// TIA Portal project "项目3" (V15)

(* hardware
DEVICE "S7-1200 station_1"  S7-1200 Station
   slot 0: "Rack_0"  S7-1200 Rack  Rack  V1.0
   slot 1: "PLC_1"  CPU 1214C DC/DC/Rly  6ES7 214-1HG40-0XB0  V4.2
DEVICE "HMI_1"  TP1500 Comfort Outdoor
   slot 0: "HMI_1"  TP1500 Comfort Outdoor  6AV2 124-0QC13-0AX0  15.0.0.0
   slot 1: "HMI_RT_1"  TP1500 Comfort Outdoor  6AV2 124-0QC13-0AX0  15.0.0.0
   slot 5: "HMI_1.IE_CP_1"  PROFINET Interface  15.0.0.0
      slot 1: "PROFINET Interface_1"  PROFINET Interface
         slot 1: "Port_1"  Port
         slot 2: "Port_2"  Port
   slot 7: "HMI_1.MPI/DP_CP_1"  MPI/DP Interface  15.0.0.0
*)

// ===== PLC "PLC_1"  CPU 1214C DC/DC/Rly =====

VAR_GLOBAL   // PLC tag table "默认变量表"
   "东西绿" AT %Q12.0 : Bool;
   "东西黄" AT %Q12.1 : Bool;
   "东西红" AT %Q12.2 : Bool;
   "东西转向" AT %Q12.3 : Bool;
   "南北绿" AT %Q12.4 : Bool;
   "南北黄" AT %Q12.5 : Bool;
   "南北红" AT %Q12.6 : Bool;
   "南北转向" AT %Q12.7 : Bool;
   "启动" AT %I4.0 : Bool;
   "System_Byte" AT %MB1 : Byte;
   "FirstScan" AT %M1.0 : Bool;
   "DiagStatusUpdate" AT %M1.1 : Bool;
   "AlwaysTRUE" AT %M1.2 : Bool;
   "AlwaysFALSE" AT %M1.3 : Bool;
   "Clock_Byte" AT %MB0 : Byte;
   "Clock_10Hz" AT %M0.0 : Bool;
   "Clock_5Hz" AT %M0.1 : Bool;
   "Clock_2.5Hz" AT %M0.2 : Bool;
   "Clock_2Hz" AT %M0.3 : Bool;
   "Clock_1.25Hz" AT %M0.4 : Bool;
   "Clock_1Hz" AT %M0.5 : Bool;
   "Clock_0.625Hz" AT %M0.6 : Bool;
   "Clock_0.5Hz" AT %M0.7 : Bool;
   "Tag_1" AT %MD100 : Time;
   "data" AT %MD50 : DInt;
   "计数器输出" AT %MD54 : DInt;
   "计数器复位" AT %MD58 : DInt;
   "Tag_2" AT %Q10.0 : Bool;
   "东西红启动" AT %M3.0 : Bool;
   "南北转向启动" AT %M3.1 : Bool;
   "南北转向闪烁启动" AT %M3.2 : Bool;
   "南北绿启动" AT %M3.3 : Bool;
   "南北闪烁启动" AT %M3.4 : Bool;
   "南北黄启动" AT %M3.5 : Bool;
   "南北红启动" AT %M3.6 : Bool;
   "东西转向启动" AT %M3.7 : Bool;
   "东西转向闪烁启动" AT %M4.0 : Bool;
   "东西绿启动" AT %M4.1 : Bool;
   "东西闪烁启动" AT %M4.2 : Bool;
   "东西黄启动" AT %M4.3 : Bool;
   "停止" AT %I4.1 : Bool;
   "启动信号1" AT %Q5.7 : Bool;
   "定时器1当前值" AT %MD4 : DInt;
   "定时器2当前值" AT %MD5 : DInt;
   "定时器1输出" AT %Q5.0 : Bool;
   "定时器2输出" AT %Q5.1 : Bool;
   "正常信号" AT %Q5.2 : Bool;
   "高峰信号" AT %Q5.3 : Bool;
   "夜间信号" AT %Q5.4 : Bool;
   "启动信号2" AT %Q5.5 : Bool;
   "启动信号3" AT %Q5.6 : Bool;
   "时间" AT %MD20 : Time_Of_Day;
   "报警信号" AT %Q13.0 : Bool;
   "夜间手动" AT %I4.4 : Bool;
   "正常手动" AT %I4.5 : Bool;
   "高峰手动" AT %I4.6 : Bool;
   "手动信号" AT %M6.0 : Bool;
   "切换手动" AT %I4.2 : Bool;
   "切换自动" AT %I4.3 : Bool;
   "报警" AT %Q1.7 : Bool;
   "1" AT %Q2.0 : Bool;
   "2" AT %Q2.1 : Bool;
   "3" AT %Q2.2 : Bool;
END_VAR

DATA_BLOCK "系统时间"   // DB1
{ S7_Optimized_Access := 'TRUE' }
VERSION : 0.1
   VAR
      当前时间 : DTL;
      ret : Int;
      设定时间 : DTL;
      ret1 : Int;
      设定时间按钮 : Bool;
   END_VAR
BEGIN
END_DATA_BLOCK

DATA_BLOCK "夜间_DB"   // DB3
{ S7_Optimized_Access := 'TRUE' }
VERSION : 0.1
// stored: InstanceOfName 夜间
"夜间"
BEGIN
END_DATA_BLOCK

DATA_BLOCK "夜间_DB_1"   // DB4
{ S7_Optimized_Access := 'TRUE' }
VERSION : 0.1
// stored: InstanceOfName 夜间
"夜间"
BEGIN
END_DATA_BLOCK

DATA_BLOCK "高峰_DB_1"   // DB6
{ S7_Optimized_Access := 'TRUE' }
VERSION : 0.1
// stored: InstanceOfName 高峰
"高峰"
BEGIN
END_DATA_BLOCK

DATA_BLOCK "正常_DB_2"   // DB8
{ S7_Optimized_Access := 'TRUE' }
VERSION : 0.1
// stored: InstanceOfName 正常
"正常"
BEGIN
END_DATA_BLOCK

// folder: System blocks/Program resources

DATA_BLOCK "计数器"   // DB2
{ S7_Optimized_Access := 'TRUE' }
AUTHOR : Simatic
FAMILY : IEC
NAME : CNTR
VERSION : 1.0
// stored: InstanceOfName IEC_COUNTER
"IEC_COUNTER"
BEGIN
END_DATA_BLOCK

DATA_BLOCK "IEC_Timer_0_DB_2"   // DB10
{ S7_Optimized_Access := 'TRUE' }
AUTHOR : Simatic
FAMILY : IEC
NAME : IEC_TMR
VERSION : 1.0
// stored: InstanceOfName IEC_TIMER
"IEC_TIMER"
BEGIN
END_DATA_BLOCK

DATA_BLOCK "IEC_Timer_0_DB_3"   // DB11
{ S7_Optimized_Access := 'TRUE' }
AUTHOR : Simatic
FAMILY : IEC
NAME : IEC_TMR
VERSION : 1.0
// stored: InstanceOfName IEC_TIMER
"IEC_TIMER"
BEGIN
END_DATA_BLOCK

// folder: (top level)

FUNCTION_BLOCK "正常"   // FB1, LAD
{ S7_Optimized_Access := 'TRUE' }
VERSION : 0.1
   VAR_INPUT
      启动 : Bool;
   END_VAR
   VAR_OUTPUT
      东西红 : Bool;
      南北转向 : Bool;
      南北绿 : Bool;
      南北黄 : Bool;
      南北红 : Bool;
      东西转向 : Bool;
      东西绿 : Bool;
      东西黄 : Bool;
   END_VAR
BEGIN

REGION Network 1: 计数
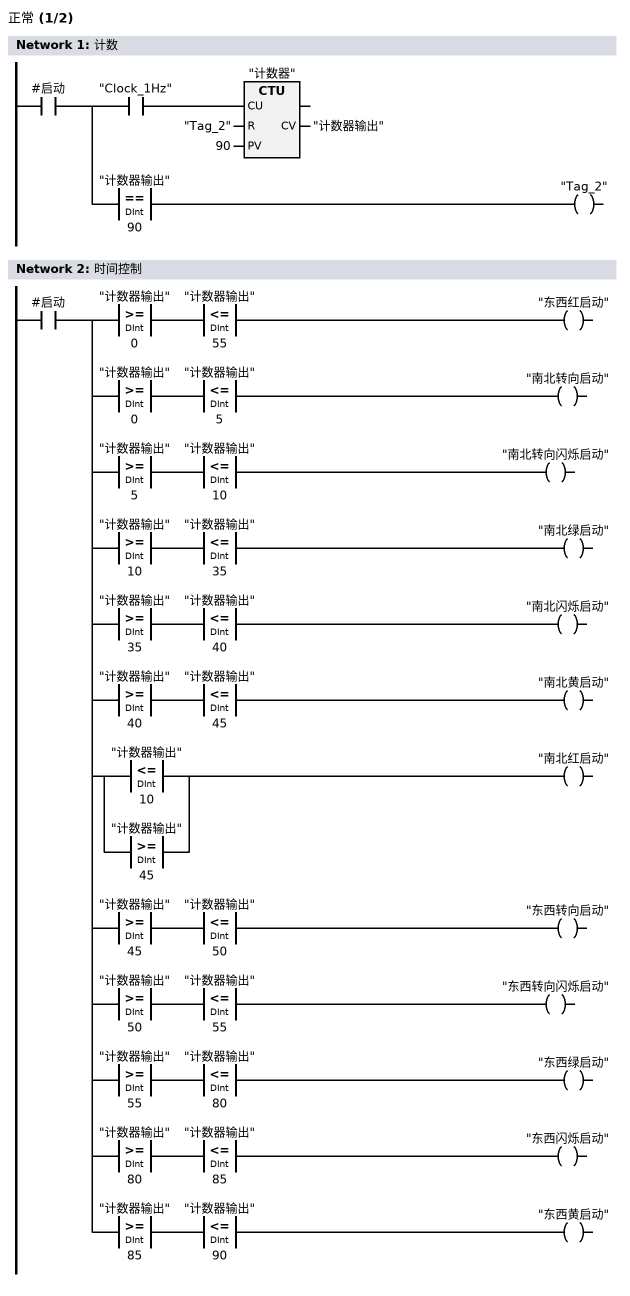
   "计数器".CTU(CU := #启动 AND "Clock_1Hz", R := "Tag_2", PV := 90, CV => "计数器输出");
   "Tag_2" := #启动 AND ("计数器输出" = 90);
END_REGION

REGION Network 2: 时间控制
   RUNG wire#powerrail
      Contact( #启动 )
      wire#w1
      { S7_Templates := "SrcType := DInt" } GE_Contact(in1 := "计数器输出", in2 := 0)
      { S7_Templates := "SrcType := DInt" } LE_Contact(in1 := "计数器输出", in2 := 55)
      Coil( "东西红启动" )
   END_RUNG
   RUNG wire#w1
      { S7_Templates := "SrcType := DInt" } GE_Contact(in1 := "计数器输出", in2 := 0)
      { S7_Templates := "SrcType := DInt" } LE_Contact(in1 := "计数器输出", in2 := 5)
      Coil( "南北转向启动" )
   END_RUNG
   RUNG wire#w1
      { S7_Templates := "SrcType := DInt" } GE_Contact(in1 := "计数器输出", in2 := 5)
      { S7_Templates := "SrcType := DInt" } LE_Contact(in1 := "计数器输出", in2 := 10)
      Coil( "南北转向闪烁启动" )
   END_RUNG
   RUNG wire#w1
      { S7_Templates := "SrcType := DInt" } GE_Contact(in1 := "计数器输出", in2 := 10)
      { S7_Templates := "SrcType := DInt" } LE_Contact(in1 := "计数器输出", in2 := 35)
      Coil( "南北绿启动" )
   END_RUNG
   RUNG wire#w1
      { S7_Templates := "SrcType := DInt" } GE_Contact(in1 := "计数器输出", in2 := 35)
      { S7_Templates := "SrcType := DInt" } LE_Contact(in1 := "计数器输出", in2 := 40)
      Coil( "南北闪烁启动" )
   END_RUNG
   RUNG wire#w1
      { S7_Templates := "SrcType := DInt" } GE_Contact(in1 := "计数器输出", in2 := 40)
      { S7_Templates := "SrcType := DInt" } LE_Contact(in1 := "计数器输出", in2 := 45)
      Coil( "南北黄启动" )
   END_RUNG
   RUNG wire#w1
      { S7_Templates := "SrcType := DInt" } LE_Contact(in1 := "计数器输出", in2 := 10)
      wire#w2
      Coil( "南北红启动" )
   END_RUNG
   RUNG wire#w1
      { S7_Templates := "SrcType := DInt" } GE_Contact(in1 := "计数器输出", in2 := 45)
   END_RUNG wire#w2
   RUNG wire#w1
      { S7_Templates := "SrcType := DInt" } GE_Contact(in1 := "计数器输出", in2 := 45)
      { S7_Templates := "SrcType := DInt" } LE_Contact(in1 := "计数器输出", in2 := 50)
      Coil( "东西转向启动" )
   END_RUNG
   RUNG wire#w1
      { S7_Templates := "SrcType := DInt" } GE_Contact(in1 := "计数器输出", in2 := 50)
      { S7_Templates := "SrcType := DInt" } LE_Contact(in1 := "计数器输出", in2 := 55)
      Coil( "东西转向闪烁启动" )
   END_RUNG
   RUNG wire#w1
      { S7_Templates := "SrcType := DInt" } GE_Contact(in1 := "计数器输出", in2 := 55)
      { S7_Templates := "SrcType := DInt" } LE_Contact(in1 := "计数器输出", in2 := 80)
      Coil( "东西绿启动" )
   END_RUNG
   RUNG wire#w1
      { S7_Templates := "SrcType := DInt" } GE_Contact(in1 := "计数器输出", in2 := 80)
      { S7_Templates := "SrcType := DInt" } LE_Contact(in1 := "计数器输出", in2 := 85)
      Coil( "东西闪烁启动" )
   END_RUNG
   RUNG wire#w1
      { S7_Templates := "SrcType := DInt" } GE_Contact(in1 := "计数器输出", in2 := 85)
      { S7_Templates := "SrcType := DInt" } LE_Contact(in1 := "计数器输出", in2 := 90)
      Coil( "东西黄启动" )
   END_RUNG
   // the same network as SCL:
   "东西红启动" := #启动 AND ("计数器输出" >= 0) AND ("计数器输出" <= 55);
   "南北转向启动" := #启动 AND ("计数器输出" >= 0) AND ("计数器输出" <= 5);
   "南北转向闪烁启动" := #启动 AND ("计数器输出" >= 5) AND ("计数器输出" <= 10);
   "南北绿启动" := #启动 AND ("计数器输出" >= 10) AND ("计数器输出" <= 35);
   "南北闪烁启动" := #启动 AND ("计数器输出" >= 35) AND ("计数器输出" <= 40);
   "南北黄启动" := #启动 AND ("计数器输出" >= 40) AND ("计数器输出" <= 45);
   "南北红启动" := #启动 AND (("计数器输出" <= 10) OR ("计数器输出" >= 45));
   "东西转向启动" := #启动 AND ("计数器输出" >= 45) AND ("计数器输出" <= 50);
   "东西转向闪烁启动" := #启动 AND ("计数器输出" >= 50) AND ("计数器输出" <= 55);
   "东西绿启动" := #启动 AND ("计数器输出" >= 55) AND ("计数器输出" <= 80);
   "东西闪烁启动" := #启动 AND ("计数器输出" >= 80) AND ("计数器输出" <= 85);
   "东西黄启动" := #启动 AND ("计数器输出" >= 85) AND ("计数器输出" <= 90);
END_REGION

REGION Network 3: 信号灯控制
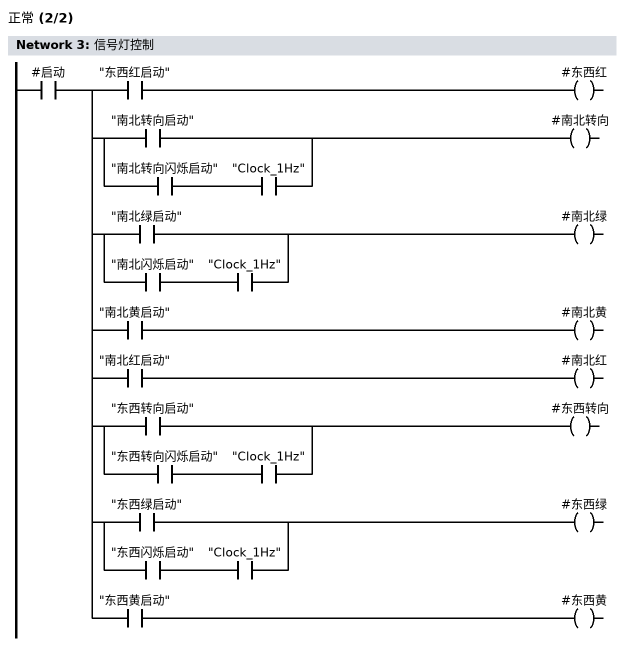
   RUNG wire#powerrail
      Contact( #启动 )
      wire#w1
      Contact( "东西红启动" )
      Coil( #东西红 )
   END_RUNG
   RUNG wire#w1
      Contact( "南北转向启动" )
      wire#w2
      Coil( #南北转向 )
   END_RUNG
   RUNG wire#w1
      Contact( "南北转向闪烁启动" )
      Contact( "Clock_1Hz" )
   END_RUNG wire#w2
   RUNG wire#w1
      Contact( "南北绿启动" )
      wire#w3
      Coil( #南北绿 )
   END_RUNG
   RUNG wire#w1
      Contact( "南北闪烁启动" )
      Contact( "Clock_1Hz" )
   END_RUNG wire#w3
   RUNG wire#w1
      Contact( "南北黄启动" )
      Coil( #南北黄 )
   END_RUNG
   RUNG wire#w1
      Contact( "南北红启动" )
      Coil( #南北红 )
   END_RUNG
   RUNG wire#w1
      Contact( "东西转向启动" )
      wire#w4
      Coil( #东西转向 )
   END_RUNG
   RUNG wire#w1
      Contact( "东西转向闪烁启动" )
      Contact( "Clock_1Hz" )
   END_RUNG wire#w4
   RUNG wire#w1
      Contact( "东西绿启动" )
      wire#w5
      Coil( #东西绿 )
   END_RUNG
   RUNG wire#w1
      Contact( "东西闪烁启动" )
      Contact( "Clock_1Hz" )
   END_RUNG wire#w5
   RUNG wire#w1
      Contact( "东西黄启动" )
      Coil( #东西黄 )
   END_RUNG
   // the same network as SCL:
   #东西红 := #启动 AND "东西红启动";
   #南北转向 := #启动 AND ("南北转向启动" OR ("南北转向闪烁启动" AND "Clock_1Hz"));
   #南北绿 := #启动 AND ("南北绿启动" OR ("南北闪烁启动" AND "Clock_1Hz"));
   #南北黄 := #启动 AND "南北黄启动";
   #南北红 := #启动 AND "南北红启动";
   #东西转向 := #启动 AND ("东西转向启动" OR ("东西转向闪烁启动" AND "Clock_1Hz"));
   #东西绿 := #启动 AND ("东西绿启动" OR ("东西闪烁启动" AND "Clock_1Hz"));
   #东西黄 := #启动 AND "东西黄启动";
END_REGION
END_FUNCTION_BLOCK

FUNCTION_BLOCK "高峰"   // FB2, LAD
{ S7_Optimized_Access := 'TRUE' }
VERSION : 0.1
   VAR_INPUT
      启动 : Bool := 0;
   END_VAR
   VAR_OUTPUT
      东西红 : Bool;
      南北转向 : Bool;
      南北绿 : Bool;
      南北黄 : Bool;
      南北红 : Bool;
      东西转向 : Bool;
      东西绿 : Bool;
      东西黄 : Bool;
   END_VAR
BEGIN

REGION Network 1: 计数
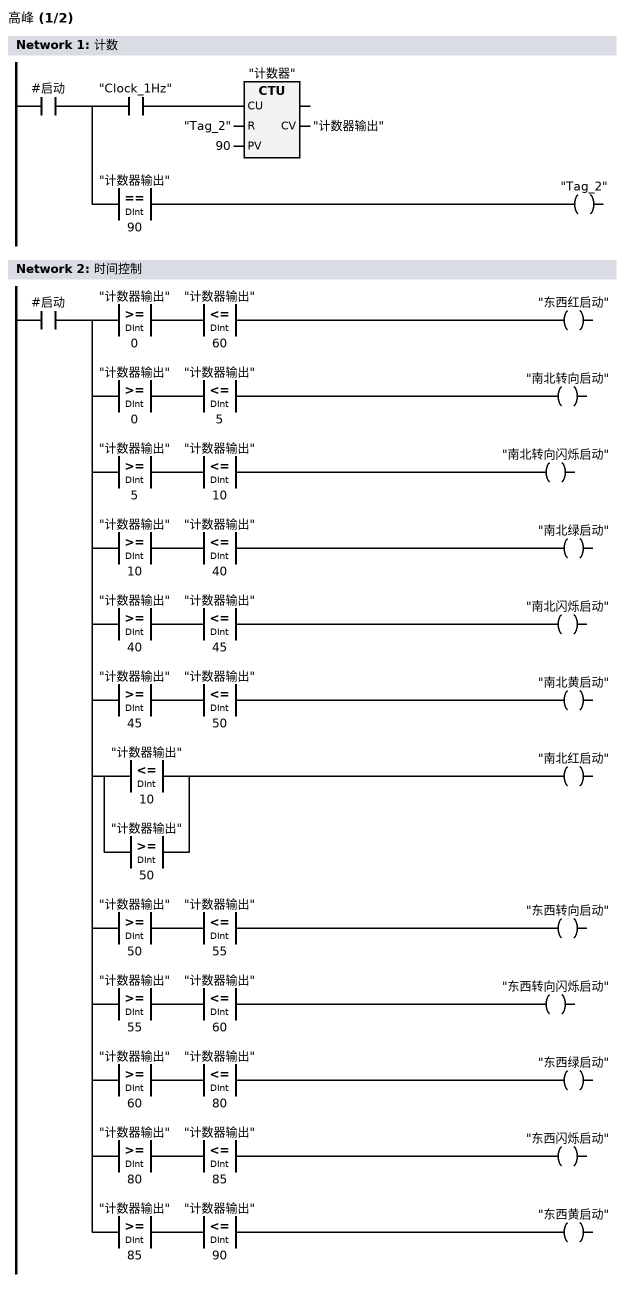
   "计数器".CTU(CU := #启动 AND "Clock_1Hz", R := "Tag_2", PV := 90, CV => "计数器输出");
   "Tag_2" := #启动 AND ("计数器输出" = 90);
END_REGION

REGION Network 2: 时间控制
   RUNG wire#powerrail
      Contact( #启动 )
      wire#w1
      { S7_Templates := "SrcType := DInt" } GE_Contact(in1 := "计数器输出", in2 := 0)
      { S7_Templates := "SrcType := DInt" } LE_Contact(in1 := "计数器输出", in2 := 60)
      Coil( "东西红启动" )
   END_RUNG
   RUNG wire#w1
      { S7_Templates := "SrcType := DInt" } GE_Contact(in1 := "计数器输出", in2 := 0)
      { S7_Templates := "SrcType := DInt" } LE_Contact(in1 := "计数器输出", in2 := 5)
      Coil( "南北转向启动" )
   END_RUNG
   RUNG wire#w1
      { S7_Templates := "SrcType := DInt" } GE_Contact(in1 := "计数器输出", in2 := 5)
      { S7_Templates := "SrcType := DInt" } LE_Contact(in1 := "计数器输出", in2 := 10)
      Coil( "南北转向闪烁启动" )
   END_RUNG
   RUNG wire#w1
      { S7_Templates := "SrcType := DInt" } GE_Contact(in1 := "计数器输出", in2 := 10)
      { S7_Templates := "SrcType := DInt" } LE_Contact(in1 := "计数器输出", in2 := 40)
      Coil( "南北绿启动" )
   END_RUNG
   RUNG wire#w1
      { S7_Templates := "SrcType := DInt" } GE_Contact(in1 := "计数器输出", in2 := 40)
      { S7_Templates := "SrcType := DInt" } LE_Contact(in1 := "计数器输出", in2 := 45)
      Coil( "南北闪烁启动" )
   END_RUNG
   RUNG wire#w1
      { S7_Templates := "SrcType := DInt" } GE_Contact(in1 := "计数器输出", in2 := 45)
      { S7_Templates := "SrcType := DInt" } LE_Contact(in1 := "计数器输出", in2 := 50)
      Coil( "南北黄启动" )
   END_RUNG
   RUNG wire#w1
      { S7_Templates := "SrcType := DInt" } LE_Contact(in1 := "计数器输出", in2 := 10)
      wire#w2
      Coil( "南北红启动" )
   END_RUNG
   RUNG wire#w1
      { S7_Templates := "SrcType := DInt" } GE_Contact(in1 := "计数器输出", in2 := 50)
   END_RUNG wire#w2
   RUNG wire#w1
      { S7_Templates := "SrcType := DInt" } GE_Contact(in1 := "计数器输出", in2 := 50)
      { S7_Templates := "SrcType := DInt" } LE_Contact(in1 := "计数器输出", in2 := 55)
      Coil( "东西转向启动" )
   END_RUNG
   RUNG wire#w1
      { S7_Templates := "SrcType := DInt" } GE_Contact(in1 := "计数器输出", in2 := 55)
      { S7_Templates := "SrcType := DInt" } LE_Contact(in1 := "计数器输出", in2 := 60)
      Coil( "东西转向闪烁启动" )
   END_RUNG
   RUNG wire#w1
      { S7_Templates := "SrcType := DInt" } GE_Contact(in1 := "计数器输出", in2 := 60)
      { S7_Templates := "SrcType := DInt" } LE_Contact(in1 := "计数器输出", in2 := 80)
      Coil( "东西绿启动" )
   END_RUNG
   RUNG wire#w1
      { S7_Templates := "SrcType := DInt" } GE_Contact(in1 := "计数器输出", in2 := 80)
      { S7_Templates := "SrcType := DInt" } LE_Contact(in1 := "计数器输出", in2 := 85)
      Coil( "东西闪烁启动" )
   END_RUNG
   RUNG wire#w1
      { S7_Templates := "SrcType := DInt" } GE_Contact(in1 := "计数器输出", in2 := 85)
      { S7_Templates := "SrcType := DInt" } LE_Contact(in1 := "计数器输出", in2 := 90)
      Coil( "东西黄启动" )
   END_RUNG
   // the same network as SCL:
   "东西红启动" := #启动 AND ("计数器输出" >= 0) AND ("计数器输出" <= 60);
   "南北转向启动" := #启动 AND ("计数器输出" >= 0) AND ("计数器输出" <= 5);
   "南北转向闪烁启动" := #启动 AND ("计数器输出" >= 5) AND ("计数器输出" <= 10);
   "南北绿启动" := #启动 AND ("计数器输出" >= 10) AND ("计数器输出" <= 40);
   "南北闪烁启动" := #启动 AND ("计数器输出" >= 40) AND ("计数器输出" <= 45);
   "南北黄启动" := #启动 AND ("计数器输出" >= 45) AND ("计数器输出" <= 50);
   "南北红启动" := #启动 AND (("计数器输出" <= 10) OR ("计数器输出" >= 50));
   "东西转向启动" := #启动 AND ("计数器输出" >= 50) AND ("计数器输出" <= 55);
   "东西转向闪烁启动" := #启动 AND ("计数器输出" >= 55) AND ("计数器输出" <= 60);
   "东西绿启动" := #启动 AND ("计数器输出" >= 60) AND ("计数器输出" <= 80);
   "东西闪烁启动" := #启动 AND ("计数器输出" >= 80) AND ("计数器输出" <= 85);
   "东西黄启动" := #启动 AND ("计数器输出" >= 85) AND ("计数器输出" <= 90);
END_REGION

REGION Network 3: 信号灯控制
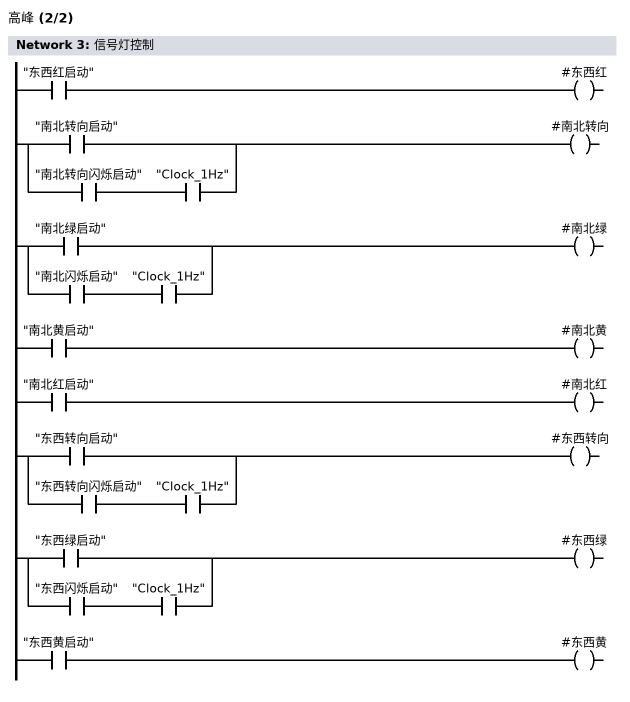
   RUNG wire#powerrail
      Contact( "东西红启动" )
      Coil( #东西红 )
   END_RUNG
   RUNG wire#powerrail
      Contact( "南北转向启动" )
      wire#w1
      Coil( #南北转向 )
   END_RUNG
   RUNG wire#powerrail
      Contact( "南北转向闪烁启动" )
      Contact( "Clock_1Hz" )
   END_RUNG wire#w1
   RUNG wire#powerrail
      Contact( "南北绿启动" )
      wire#w2
      Coil( #南北绿 )
   END_RUNG
   RUNG wire#powerrail
      Contact( "南北闪烁启动" )
      Contact( "Clock_1Hz" )
   END_RUNG wire#w2
   RUNG wire#powerrail
      Contact( "南北黄启动" )
      Coil( #南北黄 )
   END_RUNG
   RUNG wire#powerrail
      Contact( "南北红启动" )
      Coil( #南北红 )
   END_RUNG
   RUNG wire#powerrail
      Contact( "东西转向启动" )
      wire#w3
      Coil( #东西转向 )
   END_RUNG
   RUNG wire#powerrail
      Contact( "东西转向闪烁启动" )
      Contact( "Clock_1Hz" )
   END_RUNG wire#w3
   RUNG wire#powerrail
      Contact( "东西绿启动" )
      wire#w4
      Coil( #东西绿 )
   END_RUNG
   RUNG wire#powerrail
      Contact( "东西闪烁启动" )
      Contact( "Clock_1Hz" )
   END_RUNG wire#w4
   RUNG wire#powerrail
      Contact( "东西黄启动" )
      Coil( #东西黄 )
   END_RUNG
   // the same network as SCL:
   #东西红 := "东西红启动";
   #南北转向 := "南北转向启动" OR ("南北转向闪烁启动" AND "Clock_1Hz");
   #南北绿 := "南北绿启动" OR ("南北闪烁启动" AND "Clock_1Hz");
   #南北黄 := "南北黄启动";
   #南北红 := "南北红启动";
   #东西转向 := "东西转向启动" OR ("东西转向闪烁启动" AND "Clock_1Hz");
   #东西绿 := "东西绿启动" OR ("东西闪烁启动" AND "Clock_1Hz");
   #东西黄 := "东西黄启动";
END_REGION
END_FUNCTION_BLOCK

FUNCTION_BLOCK "夜间"   // FB3, LAD
{ S7_Optimized_Access := 'TRUE' }
VERSION : 0.1
   VAR_INPUT
      启动 : Bool;
   END_VAR
   VAR_OUTPUT
      南北黄启动 : Bool;
      东西黄启动 : Bool;
   END_VAR
BEGIN

REGION Network 1: 信号灯控制
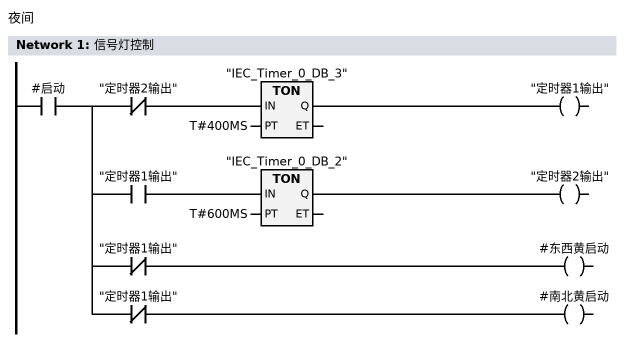
   "IEC_Timer_0_DB_3".TON(IN := #启动 AND NOT "定时器2输出", PT := T#400MS);
   "定时器1输出" := "IEC_Timer_0_DB_3".Q;
   "IEC_Timer_0_DB_2".TON(IN := #启动 AND "定时器1输出", PT := T#600MS);
   "定时器2输出" := "IEC_Timer_0_DB_2".Q;
   #东西黄启动 := #启动 AND NOT "定时器1输出";
   #南北黄启动 := #启动 AND NOT "定时器1输出";
END_REGION
END_FUNCTION_BLOCK

ORGANIZATION_BLOCK "Main"   // OB1, LAD, ProgramCycle
TITLE = "Main Program Sweep (Cycle)"
{ S7_Optimized_Access := 'TRUE' }
VERSION : 0.1
   VAR_INPUT
      Initial_Call : Bool;   // Initial call of this OB
      Remanence : Bool;   // =True, if remanent data are available
   END_VAR
   VAR_TEMP   // added for the SCL form of the ladder/FBD networks
      _w1 : Bool;
      _w2 : Bool;
      _w3 : Bool;
   END_VAR
BEGIN

REGION Network 1: 启动
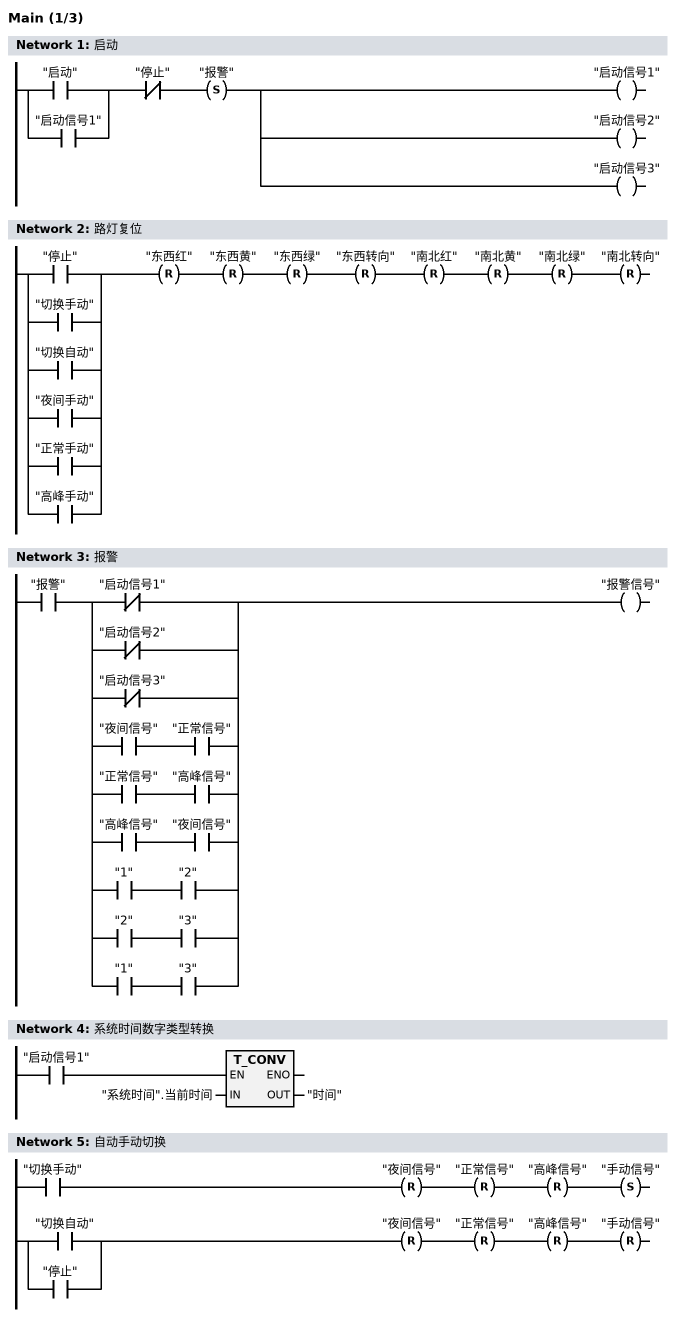
   RUNG wire#powerrail
      Contact( "启动" )
      wire#w1
      I_Contact( "停止" )
      S_Coil( "报警" )
      wire#w2
      Coil( "启动信号1" )
   END_RUNG
   RUNG wire#powerrail
      Contact( "启动信号1" )
   END_RUNG wire#w1
   RUNG wire#w2
      Coil( "启动信号2" )
   END_RUNG
   RUNG wire#w2
      Coil( "启动信号3" )
   END_RUNG
   // the same network as SCL:
   #_w1 := ("启动" OR "启动信号1") AND NOT "停止";
   IF #_w1 THEN "报警" := TRUE; END_IF;
   "启动信号1" := #_w1;
   "启动信号2" := #_w1;
   "启动信号3" := #_w1;
END_REGION

REGION Network 2: 路灯复位
   RUNG wire#powerrail
      Contact( "停止" )
      wire#w1
      R_Coil( "东西红" )
      R_Coil( "东西黄" )
      R_Coil( "东西绿" )
      R_Coil( "东西转向" )
      R_Coil( "南北红" )
      R_Coil( "南北黄" )
      R_Coil( "南北绿" )
      R_Coil( "南北转向" )
   END_RUNG
   RUNG wire#powerrail
      Contact( "切换手动" )
   END_RUNG wire#w1
   RUNG wire#powerrail
      Contact( "切换自动" )
   END_RUNG wire#w1
   RUNG wire#powerrail
      Contact( "夜间手动" )
   END_RUNG wire#w1
   RUNG wire#powerrail
      Contact( "正常手动" )
   END_RUNG wire#w1
   RUNG wire#powerrail
      Contact( "高峰手动" )
   END_RUNG wire#w1
   // the same network as SCL:
   IF "停止" OR "切换手动" OR "切换自动" OR "夜间手动" OR "正常手动" OR "高峰手动" THEN
       "东西红" := FALSE;
       "东西黄" := FALSE;
       "东西绿" := FALSE;
       "东西转向" := FALSE;
       "南北红" := FALSE;
       "南北黄" := FALSE;
       "南北绿" := FALSE;
       "南北转向" := FALSE;
   END_IF;
END_REGION

REGION Network 3: 报警
   RUNG wire#powerrail
      Contact( "报警" )
      wire#w1
      I_Contact( "启动信号1" )
      wire#w2
      Coil( "报警信号" )
   END_RUNG
   RUNG wire#w1
      I_Contact( "启动信号2" )
   END_RUNG wire#w2
   RUNG wire#w1
      I_Contact( "启动信号3" )
   END_RUNG wire#w2
   RUNG wire#w1
      Contact( "夜间信号" )
      Contact( "正常信号" )
   END_RUNG wire#w2
   RUNG wire#w1
      Contact( "正常信号" )
      Contact( "高峰信号" )
   END_RUNG wire#w2
   RUNG wire#w1
      Contact( "高峰信号" )
      Contact( "夜间信号" )
   END_RUNG wire#w2
   RUNG wire#w1
      Contact( "1" )
      Contact( "2" )
   END_RUNG wire#w2
   RUNG wire#w1
      Contact( "2" )
      Contact( "3" )
   END_RUNG wire#w2
   RUNG wire#w1
      Contact( "1" )
      Contact( "3" )
   END_RUNG wire#w2
   // the same network as SCL:
   "报警信号" := "报警" AND (NOT "启动信号1" OR NOT "启动信号2" OR NOT "启动信号3" OR ("夜间信号" AND "正常信号") OR ("正常信号" AND "高峰信号") OR ("高峰信号" AND "夜间信号") OR ("1" AND "2") OR ("2" AND "3") OR ("1" AND "3"));
END_REGION

REGION Network 4: 系统时间数字类型转换
   IF "启动信号1" THEN "时间" := T_CONV(IN := "系统时间".当前时间); END_IF;
END_REGION

REGION Network 5: 自动手动切换
   RUNG wire#powerrail
      Contact( "切换手动" )
      R_Coil( "夜间信号" )
      R_Coil( "正常信号" )
      R_Coil( "高峰信号" )
      S_Coil( "手动信号" )
   END_RUNG
   RUNG wire#powerrail
      Contact( "切换自动" )
      wire#w1
      R_Coil( "夜间信号" )
      R_Coil( "正常信号" )
      R_Coil( "高峰信号" )
      R_Coil( "手动信号" )
   END_RUNG
   RUNG wire#powerrail
      Contact( "停止" )
   END_RUNG wire#w1
   // the same network as SCL:
   IF "切换手动" THEN
       "夜间信号" := FALSE;
       "正常信号" := FALSE;
       "高峰信号" := FALSE;
       "手动信号" := TRUE;
   END_IF;
   IF "切换自动" OR "停止" THEN
       "夜间信号" := FALSE;
       "正常信号" := FALSE;
       "高峰信号" := FALSE;
       "手动信号" := FALSE;
   END_IF;
END_REGION

REGION Network 6: 手动执行不同时段程序
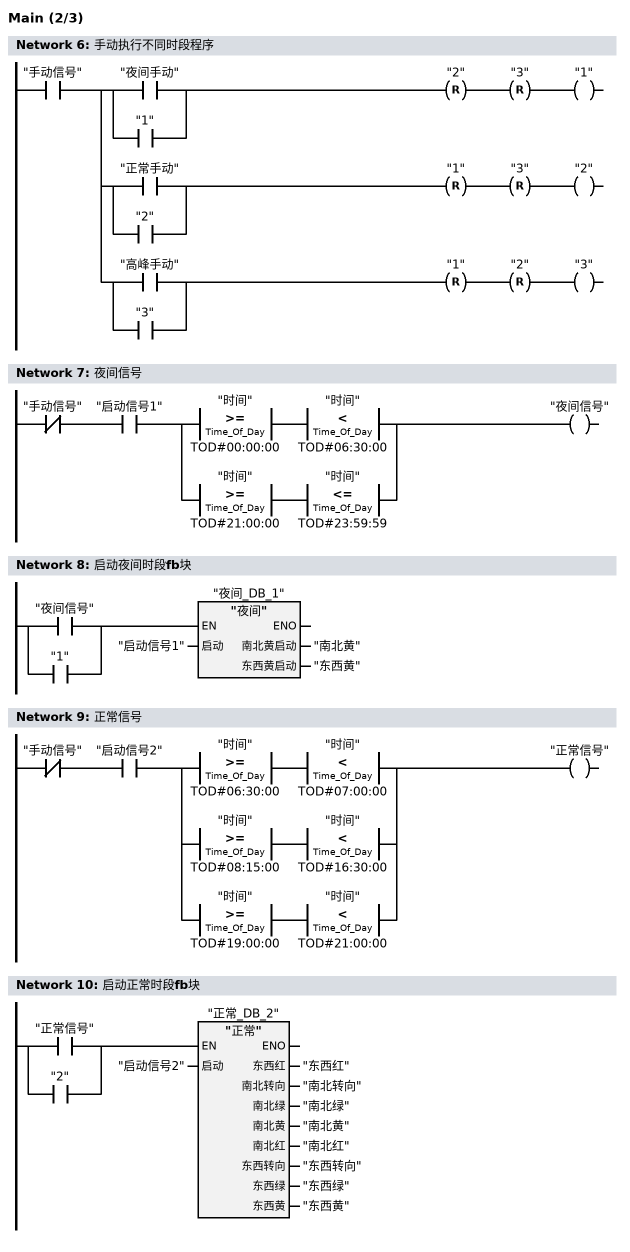
   RUNG wire#powerrail
      Contact( "手动信号" )
      wire#w1
      Contact( "夜间手动" )
      wire#w2
      R_Coil( "2" )
      R_Coil( "3" )
      Coil( "1" )
   END_RUNG
   RUNG wire#w1
      Contact( "1" )
   END_RUNG wire#w2
   RUNG wire#w1
      Contact( "正常手动" )
      wire#w3
      R_Coil( "1" )
      R_Coil( "3" )
      Coil( "2" )
   END_RUNG
   RUNG wire#w1
      Contact( "2" )
   END_RUNG wire#w3
   RUNG wire#w1
      Contact( "高峰手动" )
      wire#w4
      R_Coil( "1" )
      R_Coil( "2" )
      Coil( "3" )
   END_RUNG
   RUNG wire#w1
      Contact( "3" )
   END_RUNG wire#w4
   // the same network as SCL:
   #_w1 := "手动信号" AND ("夜间手动" OR "1");
   IF #_w1 THEN
       "2" := FALSE;
       "3" := FALSE;
   END_IF;
   "1" := #_w1;
   #_w2 := "手动信号" AND ("正常手动" OR "2");
   IF #_w2 THEN
       "1" := FALSE;
       "3" := FALSE;
   END_IF;
   "2" := #_w2;
   #_w3 := "手动信号" AND ("高峰手动" OR "3");
   IF #_w3 THEN
       "1" := FALSE;
       "2" := FALSE;
   END_IF;
   "3" := #_w3;
END_REGION

REGION Network 7: 夜间信号
   RUNG wire#powerrail
      I_Contact( "手动信号" )
      Contact( "启动信号1" )
      wire#w1
      { S7_Templates := "SrcType := Time_Of_Day" } GE_Contact(in1 := "时间", in2 := TOD#00:00:00)
      { S7_Templates := "SrcType := Time_Of_Day" } LT_Contact(in1 := "时间", in2 := TOD#06:30:00)
      wire#w2
      Coil( "夜间信号" )
   END_RUNG
   RUNG wire#w1
      { S7_Templates := "SrcType := Time_Of_Day" } GE_Contact(in1 := "时间", in2 := TOD#21:00:00)
      { S7_Templates := "SrcType := Time_Of_Day" } LE_Contact(in1 := "时间", in2 := TOD#23:59:59)
   END_RUNG wire#w2
   // the same network as SCL:
   "夜间信号" := NOT "手动信号" AND "启动信号1" AND ((("时间" >= TOD#00:00:00) AND ("时间" < TOD#06:30:00)) OR (("时间" >= TOD#21:00:00) AND ("时间" <= TOD#23:59:59)));
END_REGION

REGION Network 8: 启动夜间时段fb块
   RUNG wire#powerrail
      Contact( "夜间信号" )
      wire#w1
      "夜间_DB_1"(启动 := "启动信号1", 南北黄启动 => "南北黄", 东西黄启动 => "东西黄")
   END_RUNG
   RUNG wire#powerrail
      Contact( "1" )
   END_RUNG wire#w1
   // the same network as SCL:
   IF "夜间信号" OR "1" THEN
       "夜间_DB_1"(启动 := "启动信号1", 南北黄启动 => "南北黄", 东西黄启动 => "东西黄");   // "夜间"
   END_IF;
END_REGION

REGION Network 9: 正常信号
   RUNG wire#powerrail
      I_Contact( "手动信号" )
      Contact( "启动信号2" )
      wire#w1
      { S7_Templates := "SrcType := Time_Of_Day" } GE_Contact(in1 := "时间", in2 := TOD#06:30:00)
      { S7_Templates := "SrcType := Time_Of_Day" } LT_Contact(in1 := "时间", in2 := TOD#07:00:00)
      wire#w2
      Coil( "正常信号" )
   END_RUNG
   RUNG wire#w1
      { S7_Templates := "SrcType := Time_Of_Day" } GE_Contact(in1 := "时间", in2 := TOD#08:15:00)
      { S7_Templates := "SrcType := Time_Of_Day" } LT_Contact(in1 := "时间", in2 := TOD#16:30:00)
   END_RUNG wire#w2
   RUNG wire#w1
      { S7_Templates := "SrcType := Time_Of_Day" } GE_Contact(in1 := "时间", in2 := TOD#19:00:00)
      { S7_Templates := "SrcType := Time_Of_Day" } LT_Contact(in1 := "时间", in2 := TOD#21:00:00)
   END_RUNG wire#w2
   // the same network as SCL:
   "正常信号" := NOT "手动信号" AND "启动信号2" AND ((("时间" >= TOD#06:30:00) AND ("时间" < TOD#07:00:00)) OR (("时间" >= TOD#08:15:00) AND ("时间" < TOD#16:30:00)) OR (("时间" >= TOD#19:00:00) AND ("时间" < TOD#21:00:00)));
END_REGION

REGION Network 10: 启动正常时段fb块
   RUNG wire#powerrail
      Contact( "正常信号" )
      wire#w1
      "正常_DB_2"(启动 := "启动信号2", 东西红 => "东西红", 南北转向 => "南北转向", 南北绿 => "南北绿", 南北黄 => "南北黄", 南北红 => "南北红", 东西转向 => "东西转向", 东西绿 => "东西绿", 东西黄 => "东西黄")
   END_RUNG
   RUNG wire#powerrail
      Contact( "2" )
   END_RUNG wire#w1
   // the same network as SCL:
   IF "正常信号" OR "2" THEN
       "正常_DB_2"(启动 := "启动信号2",   // "正常"
                 东西红 => "东西红",
                 南北转向 => "南北转向",
                 南北绿 => "南北绿",
                 南北黄 => "南北黄",
                 南北红 => "南北红",
                 东西转向 => "东西转向",
                 东西绿 => "东西绿",
                 东西黄 => "东西黄");
   END_IF;
END_REGION

REGION Network 11: 高峰信号
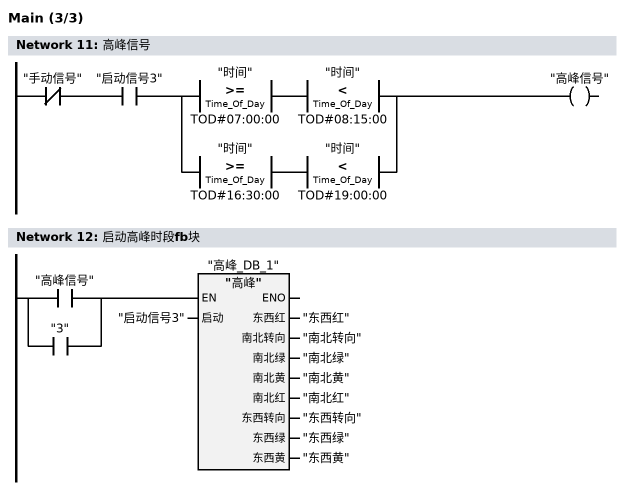
   RUNG wire#powerrail
      I_Contact( "手动信号" )
      Contact( "启动信号3" )
      wire#w1
      { S7_Templates := "SrcType := Time_Of_Day" } GE_Contact(in1 := "时间", in2 := TOD#07:00:00)
      { S7_Templates := "SrcType := Time_Of_Day" } LT_Contact(in1 := "时间", in2 := TOD#08:15:00)
      wire#w2
      Coil( "高峰信号" )
   END_RUNG
   RUNG wire#w1
      { S7_Templates := "SrcType := Time_Of_Day" } GE_Contact(in1 := "时间", in2 := TOD#16:30:00)
      { S7_Templates := "SrcType := Time_Of_Day" } LT_Contact(in1 := "时间", in2 := TOD#19:00:00)
   END_RUNG wire#w2
   // the same network as SCL:
   "高峰信号" := NOT "手动信号" AND "启动信号3" AND ((("时间" >= TOD#07:00:00) AND ("时间" < TOD#08:15:00)) OR (("时间" >= TOD#16:30:00) AND ("时间" < TOD#19:00:00)));
END_REGION

REGION Network 12: 启动高峰时段fb块
   RUNG wire#powerrail
      Contact( "高峰信号" )
      wire#w1
      "高峰_DB_1"(启动 := "启动信号3", 东西红 => "东西红", 南北转向 => "南北转向", 南北绿 => "南北绿", 南北黄 => "南北黄", 南北红 => "南北红", 东西转向 => "东西转向", 东西绿 => "东西绿", 东西黄 => "东西黄")
   END_RUNG
   RUNG wire#powerrail
      Contact( "3" )
   END_RUNG wire#w1
   // the same network as SCL:
   IF "高峰信号" OR "3" THEN
       "高峰_DB_1"(启动 := "启动信号3",   // "高峰"
                 东西红 => "东西红",
                 南北转向 => "南北转向",
                 南北绿 => "南北绿",
                 南北黄 => "南北黄",
                 南北红 => "南北红",
                 东西转向 => "东西转向",
                 东西绿 => "东西绿",
                 东西黄 => "东西黄");
   END_IF;
END_REGION
END_ORGANIZATION_BLOCK

ORGANIZATION_BLOCK "Cyclic interrupt"   // OB30, LAD, CyclicInterrupt
{ S7_Optimized_Access := 'TRUE' }
VERSION : 0.1
   VAR_INPUT
      Initial_Call : Bool;   // Initial call of this OB
      Event_Count : Int;   // Events discarded
   END_VAR
BEGIN

REGION Network 1: 调用系统时间
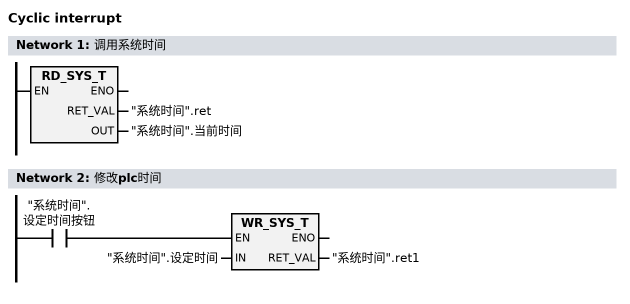
   "系统时间".ret := RD_SYS_T(OUT => "系统时间".当前时间);
END_REGION

REGION Network 2: 修改plc时间
   IF "系统时间".设定时间按钮 THEN "系统时间".ret1 := WR_SYS_T(IN := "系统时间".设定时间); END_IF;
END_REGION
END_ORGANIZATION_BLOCK

(* ===== HMI "HMI_RT_1" =====
system functions are stored by id; their names below are inferred from use
connection "HMI_连接_1": ETHERNET, S7_1200_OMS

HMI tags "默认变量表"
   "Tag_ScreenNumber" : UInt, internal
   "启动" : Bool = PLC 启动 AT %I4.0, 1 s
   "系统时间_当前时间" : DTL = PLC 系统时间.当前时间, 1 s
   "系统时间_设定时间" : DTL = PLC 系统时间.设定时间, 1 s
   "系统时间_设定时间按钮" : Bool = PLC 系统时间.设定时间按钮, 1 s
   "东西红" : Bool = PLC 东西红 AT %Q12.2, 1 s
   "东西黄" : Bool = PLC 东西黄 AT %Q12.1, 1 s
   "东西绿" : Bool = PLC 东西绿 AT %Q12.0, 1 s
   "启动信号" : Bool = PLC 启动信号1 AT %Q5.7, 1 s
   "计数器输出" : DInt = PLC 计数器输出 AT %MD54, 1 s
   "测试" : Bool = PLC 测试 AT %M4.6, 1 s
   "计数器复位" : DInt = PLC 计数器复位 AT %MD58, 1 s
   "南北红" : Bool = PLC 南北红 AT %Q12.6, 1 s
   "南北黄" : Bool = PLC 南北黄 AT %Q12.5, 1 s
   "南北绿" : Bool = PLC 南北绿 AT %Q12.4, 1 s
   "东西转向" : Bool = PLC 东西转向 AT %Q12.3, 1 s
   "南北转向" : Bool = PLC 南北转向 AT %Q12.7, 1 s
   "停止" : Bool = PLC 停止 AT %I4.1, 1 s

screen "根画面" 1280x740, template "Template_1"
   on GenerateScreen: SetTag("Tag_ScreenNumber", 1)
   Circle "圆_1" at 189,209 size 48x48
      Appearance <- "启动"
   Button "按钮_1" at 176,146 size 96x32; TextOff '启动'
      on Click: SetBit("启动")
   Button "按钮_2" at 178,296 size 96x32; TextOff '停止'
      on Click: SetBit("启动")

Template "Template_1" 1280x740
   Button "退出" at 1200,679 size 78x59; TextOff '退出'; PictureOff "ExitRuntime_TP1500_Comfort_Outdoor_TR"; PictureOn "ExitRuntime_TP1500_Comfort_Outdoor_TR"
      on Release: StopRuntime(0)
   Button "Template_Button" at 1120,679 size 78x59; TextOff 'Text'
   Button "Template_Button_1" at 1040,679 size 78x59; TextOff 'Text'
   Button "Template_Button_2" at 960,679 size 78x59; TextOff 'Text'
   Button "Template_Button_3" at 880,679 size 78x59; TextOff 'Text'
   Button "Template_Button_4" at 800,679 size 78x59; TextOff 'Text'
   Button "Template_Button_5" at 720,679 size 78x59; TextOff 'Text'
   Button "Template_Button_6" at 640,679 size 78x59; TextOff 'Text'
   Button "Template_Button_7" at 561,679 size 78x59; TextOff 'Text'
   Button "Template_Button_8" at 481,679 size 78x59; TextOff 'Text'
   Button "Template_Button_9" at 401,679 size 78x59; TextOff 'Text'
   Button "Template_Button_10" at 321,679 size 78x59; TextOff 'Text'
   Button "Template_Button_11" at 241,679 size 78x59; TextOff 'Text'
   Button "Template_Button_12" at 161,679 size 78x59; TextOff 'Text'
   Button "Template_Button_13" at 81,679 size 78x59; TextOff 'Text'
   Button "起始画面" at 1,679 size 78x59; TextOff '起始画面'; PictureOff "NavigateHome_TP1500_Comfort_Outdoor_TR"; PictureOn "NavigateHome_TP1500_Comfort_Outdoor_TR"
      on Release: ActivateScreen("根画面", 0)

screen "time" 1280x740
   DateTimeField "日期/时间域_1" at 203,113 size 548x55
      ProcessValue <- "系统时间_当前时间"
   TextField "文本域_1" at 67,113 size 77x21; Text '当前时间'
   TextField "文本域_2" at 31,195 size 113x21; Text '设定时间时间'
   DateTimeField "日期/时间域_2" at 203,195 size 548x55
      ProcessValue <- "系统时间_设定时间"
   Button "按钮_1" at 307,296 size 96x32; TextOff '设定时间'
      on Press: SetBit("系统时间_设定时间按钮")
      on Release: ResetBit("系统时间_设定时间按钮")
   Circle "圆_1" at 159,407 size 48x48
      Appearance <- "东西红"
   Circle "圆_2" at 320,407 size 48x48
      Appearance <- "东西绿"
   Circle "圆_3" at 240,407 size 48x48
      Appearance <- "东西黄"
   Circle "圆_4" at 159,483 size 48x48
      Appearance <- "启动信号"
   Circle "圆_5" at 240,483 size 48x48
      Appearance <- "启动"
   Circle "圆_6" at 320,483 size 48x48
      Appearance <- "计数器复位"
   Button "按钮_2" at 105,296 size 96x32; TextOff '启动'
      on Click: InvertBit("启动")
   Circle "圆_7" at 403,483 size 48x48
      Appearance <- "测试"
   Circle "圆_8" at 451,407 size 48x48
      Appearance <- "南北红"
   Circle "圆_9" at 530,407 size 48x48
      Appearance <- "南北黄"
   Circle "圆_10" at 609,407 size 48x48
      Appearance <- "南北绿"
   Circle "圆_11" at 451,296 size 48x48
      Appearance <- "东西转向"
   Circle "圆_12" at 609,296 size 48x48
      Appearance <- "南北转向"
   Button "按钮_3" at 211,358 size 96x32; TextOff 'stop'
      on Click: SetBit("停止"); SetBit("停止")
*)